(* PLC project KinIn_v3.project, CODESYS CODESYS V3.5 SP19 *)
(* stored: creationDateTime 2025-01-20T16:25:25.2361831, modificationDateTime 2025-01-20T16:17:39.6822999 *)

FUNCTION_BLOCK Mat_byScalar
  VAR_INPUT
    scalar : REAL;
    {attribute 'variable_length_array_original_scope' := 'Inout'}
    {attribute 'variable_length_array' := 'ARRAY[*,*] OF REAL'}
    {attribute 'Dimensions' := '2'}
    Matrix : POINTER TO REAL;
    {attribute 'variable_length_array_original_scope' := 'Inout'}
    {attribute 'variable_length_array' := 'ARRAY[*,*] OF REAL'}
    {attribute 'Dimensions' := '2'}
    MatrixByScalar : POINTER TO REAL;
  END_VAR
  VAR
    i : DINT;
    j : DINT;
  END_VAR

            FOR i:=1 TO UPPER_BOUND(Matrix,1) DO
	FOR j:=1 TO UPPER_BOUND(Matrix,2) DO
		MatrixByScalar[i,j]:=Matrix[i,j]*scalar;
	END_FOR
END_FOR
          
END_FUNCTION_BLOCK
